FUNCTION_BLOCK FuncGeneralesCortHum4
VAR_INPUT

END_VAR
VAR_OUTPUT
	s_ModeloActualTabla:STRING;
	s_ModeloEleccionTabla:STRING;
	s_JustificaParoComun:STRING;
	s_FechaInicModeloTab:STRING;
END_VAR
VAR
	Reset_Fin_Prod:BOOL;
	P_FinProduccion:BOOL;
	P_EscribirModelo:BOOL;
	sModeloEleccionTabla:STRING;
	pul_Justif_Paro:BOOL;
	Cont:INT;
	Cont1:INT;
	Cont2:INT;
	Cont3:INT;
	Cont4:INT;
END_VAR
VAR PERSISTENT 
END_VAR

//                             >>>>>>>>>>>>>>>> Modelo de la tabla <<<<<<<<<<<<<<<<<

//Fin de producción 		
IF P_FinProduccion THEN 
Fin_Produccion();
END_IF;
IF P_EscribirModelo THEN 
	Inicio_Nuevo_Modelo();
END_IF


Direccionamiento_variables_com();

ACTION Direccionamiento_variables_com:
	//                           	>>>>>>>>>>>>>>>>>>>>>>>>>>>>      STRING  <<<<<<<<<<<<<<<<<<<<<<<<<<<<<<<<
    Var_Com_CH4_MulDis.aStringCom[80] := s_ModeloActualTabla;
	Var_Com_CH4_MulDis.aStringCom[81] := s_ModeloEleccionTabla;
	Var_Com_CH4_MulDis.aStringCom[82] := s_FechaInicModeloTab;
	Var_Com_CH4_MulDis.aStringCom[83] := s_FechaInicModeloTab;
END_ACTION

METHOD Fin_Produccion : BOOL
VAR_INPUT	
END_VAR
var
	Puls_Fin_Produccion:BOOL;	
END_VAR
//Llamada a la función de fin de producción de Corte húmedo 4
FuncParoNodoCorteH4Remote1.Funci_CortHum4.Fin_Produccion();



s_ModeloActualTabla:= 'Sin modelo de pieza';
//	FechaInicModeloTab:= 'Sin modelo de pieza';
s_ModeloEleccionTabla:= 'Sin modelo de pieza';
END_METHOD

METHOD Inicio_Nuevo_Modelo : BOOL
VAR_INPUT
END_VAR
VAR
END_VAR

// Envías la fecha de inicio modelo de tabla 
s_FechaInicModeloTab:=Fecha_PLC.Mes_Dia_Hora_Min_Real;

//Envías el modelo de la tabla de la variable preelección  
s_ModeloActualTabla:=s_ModeloEleccionTabla;
END_METHOD

END_FUNCTION_BLOCK

(* stored: Version 1.1.0.1, ProductVersion 3.1.4024.12
   POU FuncGeneralesCortHum4: Id {497e5837-1248-4be6-b299-ef2f796ca598}, SpecialFunc None
   Action Direccionamiento_variables_com: Id {4cb71bcf-b2bc-47a4-9856-c8a61ddd8fd6}
   Method Fin_Produccion: Id {9cb73819-1a22-40e9-a2d8-887e90cd0ccd}
   Method Inicio_Nuevo_Modelo: Id {71048897-297a-4d08-9c81-7534270db74f} *)
